FUNCTION_BLOCK FB_Fallible_Test EXTENDS TcUnit.FB_TestSuite


TestGetErrorExpectErrorStatus();

TestGetErrorMsgExpectErrorMsg();


METHOD PRIVATE TestGetErrorExpectErrorStatus
VAR
    fbFallible : FB_Fallible;
END_VAR

TEST('TestGetErrorExpectErrorStatus');

// Test fixture

// Subject Under Test
AssertFalse(
    Condition := fbFallible.GetError(),
    Message := 'Expected GetError to be false, but it was true.'
);

TEST_FINISHED();
END_METHOD


METHOD PRIVATE TestGetErrorMsgExpectErrorMsg
VAR
    fbFallible : FB_Fallible;
END_VAR

TEST('TestGetErrorMsgExpectErrorMsg');

// Test fixture

// Subject Under Test
AssertTrue(
    Condition := fbFallible.GetErrorMsg() = '',
    Message := 'Expected GetErrorMsg to return an empty string, but it was not empty.'
);

TEST_FINISHED();
END_METHOD

END_FUNCTION_BLOCK

(* stored: Version 1.1.0.1
   POU FB_Fallible_Test: Id {8cba201b-995e-4a53-ab27-125a677e950d}, SpecialFunc None
   Method TestGetErrorExpectErrorStatus: Id {7af2bd4d-126f-48e4-a5e0-0cfb44d45ac2}
   Method TestGetErrorMsgExpectErrorMsg: Id {b950e335-0166-4227-9f34-82d4d878960b} *)
